FUNCTION_BLOCK FB_Enclosure
VAR
	// =============== Table clamping  ================================================
	pbTableWest				AT %I* : BOOL;
	pbTableEast				AT %I* : BOOL;

	pbTableWestLast: BOOL;
	pbTableEastLast: BOOL;
	cylinderTableWest		AT %Q* : BOOL := FALSE;
	cylinderTableEast		AT %Q* : BOOL := FALSE;
	
	// Door
	openCloseDoor				AT %Q* : BOOL;
	enableRollingDoor 			AT %Q* : BOOL := TRUE;
	doorIsOpen					AT %I* : BOOL;
	doorTimer				: TON;
	startTimer: BOOL;
	
	dustCollectionOn : BOOL;
END_VAR

// Reverts door to pushbutton operation once 0.5s has passed
IF startTimer THEN
	doorTimer(IN:=TRUE, PT:=T#500MS);
END_IF

IF doorTimer.Q THEN
	openCloseDoor := FALSE;
	doorTimer(IN:=FALSE);
	startTimer := FALSE;
END_IF

//Opens and closes door
METHOD Rolling_Door_HMI_Operation
VAR_INPUT
END_VAR
openCloseDoor := TRUE;
startTimer := TRUE;
END_METHOD

METHOD Table_Clamp_Control_HMI
VAR_INPUT
	eastTableLock : BOOL;
	westTableLock : BOOL;
END_VAR
cylinderTableWest := westTableLock;
cylinderTableEast := eastTableLock;
END_METHOD

METHOD Table_Clamp_Control_Pushbutton
VAR_INPUT
END_VAR
IF pbTableWest AND NOT pbTableWestLast THEN
	cylinderTableWest := NOT cylinderTableWest;
END_IF

pbTableWestLast := pbTableWest;

IF pbTableEast AND NOT pbTableEastLast THEN
	cylinderTableEast := NOT cylinderTableEast;
END_IF

pbTableEastLast := pbTableEast;
END_METHOD

END_FUNCTION_BLOCK

(* stored: Version 1.1.0.1, ProductVersion 3.1.4024.12
   POU FB_Enclosure: Id {99e77f18-d45f-4cfb-8b39-3900b2091860}, SpecialFunc None
   Method Rolling_Door_HMI_Operation: Id {30d6fe7d-957f-4531-95df-ed9ab926cc71}
   Method Table_Clamp_Control_HMI: Id {e853bb91-f390-4b22-b7cb-ad932ff4f252}
   Method Table_Clamp_Control_Pushbutton: Id {78b6b307-6e7b-4cd9-b1f5-bb2aefea736b} *)
